// TIA Portal V16 export
// export: Created 2025-05-24T14:08:00.039312Z, ExportSetting WithDefaults, DisplayName Totally Integrated Automation Portal, DisplayVersion V16, DisplayName TIA Portal Version Control Interface, DisplayVersion V16, DisplayName TIA Portal Openness, DisplayVersion V16, DisplayName STEP 7 Professional, DisplayVersion V16, DisplayName STEP 7 Safety, DisplayVersion V16, DisplayName WinCC Advanced, DisplayVersion V16
DATA_BLOCK "MC_Move_1"   // DB76
VERSION : 0.1
// stored: AutoNumber true, InstanceOfName MC_Move, InstanceOfType FB
"MC_Move"
   // VAR_INPUT
   //    Start : Bool;
   //    "Desired Position" : Real;
   //    "Speed (50-75%)" : Int;
   //    "Brake on Position" : Bool;
   //    Acceleration : Real;
   //    Deacceleration : Real;
   //    "Drive Ready" : Bool;
   //    "Drive On Position" : Bool;
   //    "Brake Time" : Time;
   //    "Safety OK" : Bool;
   // END_VAR
   // VAR_OUTPUT
   //    Go : Bool;
   //    "Desired Position Out" : Real;
   //    "Speed Output" : Int;
   //    "Acceleration Out" : Real;
   //    "Deacceleration Out" : Real;
   //    "Brake Out" : Bool;
   // END_VAR
BEGIN
END_DATA_BLOCK
